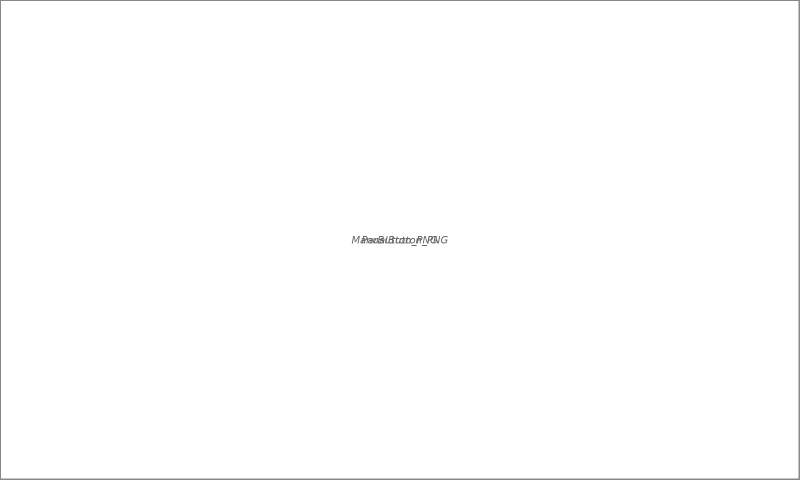
VISUALIZATION Settings_PNG  // 800x480
    Frame (0,0 800x480)
        shows ManualButton_PNG(bCmdManual := GVL_HMI.bCmdManual)
    Frame (0,0 800x480)
        shows ParButton_PNG(bCmdParameter := GVL_HMI.bCmdParemeter)
END_VISUALIZATION

(* stored: Version 1.1.0.1, ProductVersion 3.1.4024.11
   Visu Settings_PNG: Id {902dec27-9ce0-460e-9363-33508825ca96} *)
